PROGRAM P_Demo_F_BA_SetSchedulerEntry
VAR
    argTEntryTime                  : TIME                           := T#5S; // tEntryTime
    argUEntryValue                 : U_BA_ClassValue               ; // uEntryValue
    ioStEntry                      : ST_BA_SchedEntry; // stEntry 双向
    fnReturn                       : BOOL; // 返回值
END_VAR

// =============================================================================
// Tc3_BA2_Common.F_BA_SetSchedulerEntry 演示程序
// =============================================================================
// 场景：在调度数组里插入一条"每周一上午 8:00 启动空调 + 持续 10 小时 + 设定温度 22℃"的条目。
//
// 价值：一行 FC 替代手写多字段赋值；保证字段一致性（无遗漏字段）。
//
// 验证：登录 PLC 后，按例程内变量在线写值；监视输出 / 返回值，结合 §1 功能
//       简述的预期行为对照（详见配套 .md 文档 §7 业务场景）。
//
// 验证步骤：
//   1. 右键 PLC 项目下 POUs 文件夹 → Add → Existing Item → 选本 .TcPOU 文件
//   2. 引用 Tc3_BA2_Common（References → Add library）
//   3. 编译 → 登录 → 运行；按上方『验证』指引在线写值观察
// =============================================================================

fnReturn := F_BA_SetSchedulerEntry(
    tEntryTime               := argTEntryTime,
    uEntryValue              := argUEntryValue,
    stEntry                  := ioStEntry
);

END_PROGRAM

(* stored: Version 1.1.0.1, ProductVersion 3.1.4024.5
   POU P_Demo_F_BA_SetSchedulerEntry: Id {2cd001d3-a5fc-5309-9174-f17c840394fe}, SpecialFunc None *)
